// TIA Portal V18 export
TYPE "UDT_AHUsMode"
// stored: IsFailsafeCompliant false
   STRUCT
      cPreviousOne { S7_SetPoint := 'True'} : Array[1..3] of Byte;
      cActual { S7_SetPoint := 'True'} : Array[1..3] of Byte;   // Поточний/Актуальний режим роботи
      cTarget { S7_SetPoint := 'True'} : Array[1..3] of Byte;   // Вибраний режим роботи, але ще не дійшли до нього
      cPreselectedOpModePLC : Array[1..3] of Byte;   // Вибор режиму роботи з PLC. 0-Protection/1-economy/2-PreComfort/3-Comfort/4-Auto
      cSchedulerTargetUnitOpMode : Array[1..3] of Byte;
      cPreselectedOpMode : Array[1..3] of Byte;   // Вибор режиму роботи з Фызичного перемикача на шафы. 0-Protection/1-economy/2-PreComfort/3-Comfort/4-Auto
   END_STRUCT;
END_TYPE
